KUKA KRL data list: AtualizaVariaveis.dat

&ACCESS RV1
DEFDAT AtualizaVariaveis

ENDDAT
